Staubli VAL3: remMovHandler.pgx

program remMovHandler()
  local bool LbError
  local string LsCommandString
  local string LsCubeValsIOC
  local string LsCylValsIOC
  local string LsESTOPIOC
  local string LsError
  local string LsIOCCommand
  local string LsJointValsIOC
  local string LsLength
  local string LsResponse
  local string LsSphValsIOC
  local string LsTCPValsIOC
begin
  // Handle movement commands
  //
  while true
    if sRemMotionCmd!=""
      bRemMotionBusy=true
      switch sRemMotionCmd
        case "MOVXYZ"
          if nMovArgs==6
            call remMovXYZ(sIOCCommand,LsResponse)
          else
            call remErrArgs(sRemMotionCmd,nMovArgs,6,LsResponse)
          endIf
        break
        case "MOVAZELRA"
          if nMovArgs==3
            call remMovAZELRA(sIOCCommand,LsResponse)
          else
            call remErrArgs(sRemMotionCmd,nMovArgs,3,LsResponse)
          endIf
        break
        case "MOVAXIS"
          if nMovArgs==2
            call remMovAxis(sIOCCommand,LsResponse)
          else
            call remErrArgs(sRemMotionCmd,nMovArgs,2,LsResponse)
          endIf
        break
        case "MOVSPHAXIS"
          if nMovArgs==2
            call remMovSphAxis(sIOCCommand,LsResponse)
          else
            call remErrArgs(sRemMotionCmd,nMovArgs,2,LsResponse)
          endIf
        break
        case "MOVJOINT"
          if nMovArgs==6
            call remMovJoint(sIOCCommand,LsResponse)
          else
            call remErrArgs(sRemMotionCmd,nMovArgs,6,LsResponse)
          endIf
        break
        case "MOVJOINTAXIS"
          if nMovArgs==2
            call remMovJointAxis(sIOCCommand,LsResponse)
          else
            call remErrArgs(sRemMotionCmd,nMovArgs,2,LsResponse)
          endIf
        break
        default
          call remErrCmd(sRemMotionCmd,LsResponse)
        break
      endSwitch
      if len(LsResponse)>0
        call iocWriteBack(LsResponse)
      endIf
      sRemMotionCmd=""
      sIOCCommand=""
      nMovArgs=0
      bRemMotionBusy=false
    endIf
    delay(0)
  endWhile
end
